FUNCTION_BLOCK Spreader EXTENDS OperationalParticleSet
  VAR
    lSpuriousLoweredEndAB : SpuriousLoweredEnd;
    lSpuriousLoweredEndCD : SpuriousLoweredEnd;
    lTwistlocksReadyState : BOOL;
    lTwistlocksReadyStateCandidate : BOOL;
    lTwistlocksCurrentState : t_lock_state;
    lTwistlocksCurrentStateCandidate : t_lock_state;
    lTwistlocksEnabled : BOOL;
    lTwistlocksEnabledCandidate : BOOL;
    lTwistlockACurrentState : t_lock_state;
    lTwistlockALoweredState : ValueObjectBool;
    lTwistlockAReadyState : BOOL;
    lTwistlockACurrentStateCandidate : t_lock_state;
    lTwistlockALoweredStateCandidate : BOOL;
    lTwistlockAReadyStateCandidate : BOOL;
    lTwistlockBCurrentState : t_lock_state;
    lTwistlockBLoweredState : ValueObjectBool;
    lTwistlockBReadyState : BOOL;
    lTwistlockBCurrentStateCandidate : t_lock_state;
    lTwistlockBLoweredStateCandidate : BOOL;
    lTwistlockBReadyStateCandidate : BOOL;
    lTwistlockCCurrentState : t_lock_state;
    lTwistlockCLoweredState : ValueObjectBool;
    lTwistlockCReadyState : BOOL;
    lTwistlockCCurrentStateCandidate : t_lock_state;
    lTwistlockCLoweredStateCandidate : BOOL;
    lTwistlockCReadyStateCandidate : BOOL;
    lTwistlockDCurrentState : t_lock_state;
    lTwistlockDLoweredState : ValueObjectBool;
    lTwistlockDReadyState : BOOL;
    lTwistlockDCurrentStateCandidate : t_lock_state;
    lTwistlockDLoweredStateCandidate : BOOL;
    lTwistlockDReadyStateCandidate : BOOL;
  END_VAR

            ;
          

METHOD initialize
                  lSpuriousLoweredEndAB.Name := 'AB';
lSpuriousLoweredEndAB.Context REF= gSystemApollo.Lift.InputObject;
lSpuriousLoweredEndAB.PositionA REF= gSystemApollo.CANOpenMasterDriveApollo.WinchAngleA.PositionObject;
lSpuriousLoweredEndAB.PositionB REF= gSystemApollo.CANOpenMasterDriveApollo.WinchAngleB.PositionObject;
lSpuriousLoweredEndAB.TwistlockALoweredState REF= lTwistlockALoweredState;
lSpuriousLoweredEndAB.TwistlockALoweredStateCandidate REF= lTwistlockALoweredStateCandidate;
lSpuriousLoweredEndAB.TwistlockBLoweredState REF= lTwistlockBLoweredState;
lSpuriousLoweredEndAB.TwistlockBLoweredStateCandidate REF= lTwistlockBLoweredStateCandidate;
registerOperational(ADR(lSpuriousLoweredEndAB));

lSpuriousLoweredEndCD.Name := 'CD';
lSpuriousLoweredEndCD.Context REF= gSystemApollo.Lift.InputObject;
lSpuriousLoweredEndCD.PositionA REF= gSystemApollo.CANOpenMasterDriveApollo.WinchAngleC.PositionObject;
lSpuriousLoweredEndCD.PositionB REF= gSystemApollo.CANOpenMasterDriveApollo.WinchAngleD.PositionObject;
lSpuriousLoweredEndCD.TwistlockALoweredState REF= lTwistlockCLoweredState;
lSpuriousLoweredEndCD.TwistlockALoweredStateCandidate REF= lTwistlockCLoweredStateCandidate;
lSpuriousLoweredEndCD.TwistlockBLoweredState REF= lTwistlockDLoweredState;
lSpuriousLoweredEndCD.TwistlockBLoweredStateCandidate REF= lTwistlockDLoweredStateCandidate;
registerOperational(ADR(lSpuriousLoweredEndCD));

lTwistlockALoweredState.initializeValueObjectOp(OpSelf,'TwstALow','Twistlock A lowered','',cValueStyleConfigurable);
lTwistlockBLoweredState.initializeValueObjectOp(OpSelf,'TwstBLow','Twistlock B lowered','',cValueStyleConfigurable);
lTwistlockCLoweredState.initializeValueObjectOp(OpSelf,'TwstCLow','Twistlock C lowered','',cValueStyleConfigurable);
lTwistlockDLoweredState.initializeValueObjectOp(OpSelf,'TwstDLow','Twistlock D lowered','',cValueStyleConfigurable);

SUPER^.initialize();
SubSystem := cSubsystemSpreader;

                
END_METHOD

METHOD operator
                  lTwistlockACurrentStateCandidate := gSystemApollo.CANOpenMasterDriveApollo.Spreader.TwistlockACurrentState;
lTwistlockALoweredStateCandidate := gSystemApollo.CANOpenMasterDriveApollo.Spreader.TwistlockALoweredState;
lTwistlockAReadyStateCandidate := gSystemApollo.CANOpenMasterDriveApollo.Spreader.TwistlockAReadyState;

lTwistlockACurrentState := lTwistlockACurrentStateCandidate;
lTwistlockALoweredState.Value := lTwistlockALoweredStateCandidate;
lTwistlockAReadyState := lTwistlockAReadyStateCandidate;

lTwistlockBCurrentStateCandidate := gSystemApollo.CANOpenMasterDriveApollo.Spreader.TwistlockBCurrentState;
lTwistlockBLoweredStateCandidate := gSystemApollo.CANOpenMasterDriveApollo.Spreader.TwistlockBLoweredState;
lTwistlockBReadyStateCandidate := gSystemApollo.CANOpenMasterDriveApollo.Spreader.TwistlockBReadyState;

lTwistlockBCurrentState := lTwistlockBCurrentStateCandidate;
lTwistlockBLoweredState.Value := lTwistlockBLoweredStateCandidate;
lTwistlockBReadyState := lTwistlockBReadyStateCandidate;

lTwistlockCCurrentStateCandidate := gSystemApollo.CANOpenMasterDriveApollo.Spreader.TwistlockCCurrentState;
lTwistlockCLoweredStateCandidate := gSystemApollo.CANOpenMasterDriveApollo.Spreader.TwistlockCLoweredState;
lTwistlockCReadyStateCandidate := gSystemApollo.CANOpenMasterDriveApollo.Spreader.TwistlockCReadyState;

lTwistlockCCurrentState := lTwistlockCCurrentStateCandidate;
lTwistlockCLoweredState.Value := lTwistlockCLoweredStateCandidate;
lTwistlockCReadyState := lTwistlockCReadyStateCandidate;

lTwistlockDCurrentStateCandidate := gSystemApollo.CANOpenMasterDriveApollo.Spreader.TwistlockDCurrentState;
lTwistlockDLoweredStateCandidate := gSystemApollo.CANOpenMasterDriveApollo.Spreader.TwistlockDLoweredState;
lTwistlockDReadyStateCandidate := gSystemApollo.CANOpenMasterDriveApollo.Spreader.TwistlockDReadyState;

lTwistlockDCurrentState := lTwistlockDCurrentStateCandidate;
lTwistlockDLoweredState.Value := lTwistlockDLoweredStateCandidate;
lTwistlockDReadyState := lTwistlockDReadyStateCandidate;

lTwistlocksReadyStateCandidate := gSystemApollo.CANOpenMasterDriveApollo.Spreader.TwistlocksReadyState;
lTwistlocksReadyState := lTwistlocksReadyStateCandidate;

lTwistlocksCurrentStateCandidate := gSystemApollo.CANOpenMasterDriveApollo.Spreader.TwistlocksCurrentState;
lTwistlocksCurrentState := lTwistlocksCurrentStateCandidate;
IF (lTwistlocksCurrentState=t_lock_state.cLockStateNone) THEN
	lTwistlocksCurrentState := t_lock_state.cLockStatePartial;
END_IF

SUPER^.operator();

lTwistlocksEnabledCandidate := gSystemApollo.CANOpenMasterDriveApollo.Spreader.TwistlocksEnabled;
lTwistlocksEnabled := ((lTwistlocksEnabledCandidate) OR
	((lTwistlockALoweredState.Value) AND
	(lTwistlockBLoweredState.Value) AND
	(lTwistlockCLoweredState.Value) AND
	(lTwistlockDLoweredState.Value)));
		
                
END_METHOD

PROPERTY TwistlockACurrentState : t_lock_state
GET
                    TwistlockACurrentState := lTwistlockACurrentState;

                  
END_GET
END_PROPERTY

PROPERTY TwistlockALoweredState : BOOL
GET
                    TwistlockALoweredState := lTwistlockALoweredState.Value;

                  
END_GET
END_PROPERTY

PROPERTY TwistlockALoweredStateObject : REFERENCE TO ValueObjectBool
GET
                    TwistlockALoweredStateObject REF= lTwistlockALoweredState;

                  
END_GET
END_PROPERTY

PROPERTY TwistlockAReadyState : BOOL
GET
                    TwistlockAReadyState := lTwistlockAReadyState;

                  
END_GET
END_PROPERTY

PROPERTY TwistlockBCurrentState : t_lock_state
GET
                    TwistlockBCurrentState := lTwistlockBCurrentState;

                  
END_GET
END_PROPERTY

PROPERTY TwistlockBLoweredState : BOOL
GET
                    TwistlockBLoweredState := lTwistlockBLoweredState.Value;

                  
END_GET
END_PROPERTY

PROPERTY TwistlockBLoweredStateObject : REFERENCE TO ValueObjectBool
GET
                    TwistlockBLoweredStateObject REF= lTwistlockBLoweredState;

                  
END_GET
END_PROPERTY

PROPERTY TwistlockBReadyState : BOOL
GET
                    TwistlockBReadyState := lTwistlockBReadyState;

                  
END_GET
END_PROPERTY

PROPERTY TwistlockCCurrentState : t_lock_state
GET
                    TwistlockCCurrentState := lTwistlockCCurrentState;

                  
END_GET
END_PROPERTY

PROPERTY TwistlockCLoweredState : BOOL
GET
                    TwistlockCLoweredState := lTwistlockCLoweredState.Value;

                  
END_GET
END_PROPERTY

PROPERTY TwistlockCLoweredStateObject : REFERENCE TO ValueObjectBool
GET
                    TwistlockCLoweredStateObject REF= lTwistlockCLoweredState;

                  
END_GET
END_PROPERTY

PROPERTY TwistlockCReadyState : BOOL
GET
                    TwistlockCReadyState := lTwistlockCReadyState;

                  
END_GET
END_PROPERTY

PROPERTY TwistlockDCurrentState : t_lock_state
GET
                    TwistlockDCurrentState := lTwistlockDCurrentState;

                  
END_GET
END_PROPERTY

PROPERTY TwistlockDLoweredState : BOOL
GET
                    TwistlockDLoweredState := lTwistlockDLoweredState.Value;

                  
END_GET
END_PROPERTY

PROPERTY TwistlockDLoweredStateObject : REFERENCE TO ValueObjectBool
GET
                    TwistlockDLoweredStateObject REF= lTwistlockDLoweredState;

                  
END_GET
END_PROPERTY

PROPERTY TwistlockDReadyState : BOOL
GET
                    TwistlockDReadyState := lTwistlockDReadyState;

                  
END_GET
END_PROPERTY

PROPERTY TwistlocksCurrentState : t_lock_state
GET
                    TwistlocksCurrentState := lTwistlocksCurrentState;

                  
END_GET
END_PROPERTY

PROPERTY TwistlocksEnabled : BOOL
GET
                    TwistlocksEnabled := lTwistlocksEnabled;

                  
END_GET
END_PROPERTY

PROPERTY TwistlocksReadyState : BOOL
GET
                    TwistlocksReadyState := lTwistlocksReadyState;

                  
END_GET
END_PROPERTY

PROPERTY TypeToken : t_medium_string
GET
                    TypeToken := 'Spreader';
                  
END_GET
END_PROPERTY
END_FUNCTION_BLOCK

FUNCTION_BLOCK SpuriousLoweredEnd EXTENDS NonOperationalParticleSet
  VAR
    lEnable : BOOL := TRUE;
    lContext : REFERENCE TO ValueObjectPercentage;
    lPositionA : REFERENCE TO ValueObjectPercentage;
    lPositionB : REFERENCE TO ValueObjectPercentage;
    lPositionLimit : t_percentage := 0.05;  (* machine height dependent *)
    lContextReset : t_percentage := 0.05;
    lPosition : t_percentage;
    lResetPosition : t_percentage;
    lAllowAdditionalMovement : BOOL;
    lTwistlockALoweredState : REFERENCE TO ValueObjectBool;
    lTwistlockALoweredStateCandidate : REFERENCE TO BOOL;
    lTwistlockBLoweredState : REFERENCE TO ValueObjectBool;
    lTwistlockBLoweredStateCandidate : REFERENCE TO BOOL;
  END_VAR

            ;
          

METHOD operator
                  SUPER^.operator();

IF (NOT(lEnable)) THEN
	RETURN;
END_IF

// robustness measures:
// traveling and one false/on (sensor false positive or container moves): masked until lowered to limit, further upon context reset
// lowering and one false/off (sensor fails to detect): allows further lowering to limit, warning as further upon context reset possible
// lowered but chassis/stack movement or signaled too early or pulse raised: masked until lowered to limit

// average is considered more robust than per corner specific 
lPosition := (lPositionA.Value + lPositionB.Value) / 2.0;

// foobar error handling notification

IF ((lTwistlockALoweredStateCandidate) AND (lTwistlockBLoweredStateCandidate)) THEN
	lAllowAdditionalMovement := ((lResetPosition - lPosition) < lPositionLimit);

	lTwistlockALoweredState.Value := NOT(lAllowAdditionalMovement);
	lTwistlockBLoweredState.Value := NOT(lAllowAdditionalMovement);

	RETURN;
END_IF
	
IF (((NOT(lTwistlockALoweredStateCandidate)) AND (lTwistlockBLoweredStateCandidate)) OR	
	((NOT(lTwistlockBLoweredStateCandidate)) AND (lTwistlockALoweredStateCandidate))) THEN
	IF (lContext.Value>=lContextReset) THEN		
		lResetPosition := lPosition;
	END_IF

	lAllowAdditionalMovement := ((lResetPosition - lPosition) < lPositionLimit);

	lTwistlockALoweredState.Value := NOT(lAllowAdditionalMovement);
	lTwistlockBLoweredState.Value := NOT(lAllowAdditionalMovement);
	
	RETURN;
END_IF

lResetPosition := lPosition;

lTwistlockALoweredState.Value := lTwistlockALoweredStateCandidate;
lTwistlockBLoweredState.Value := lTwistlockBLoweredStateCandidate;

                
END_METHOD

PROPERTY Context : REFERENCE TO ValueObjectPercentage
GET
                    Context ref= lContext;
                  
END_GET
SET
                    lContext ref= Context;
                  
END_SET
END_PROPERTY

PROPERTY ContextReset : t_percentage
GET
                    ContextReset := lContextReset;
                  
END_GET
SET
                    lContextReset := ContextReset;
                  
END_SET
END_PROPERTY

PROPERTY PositionA : REFERENCE TO ValueObjectPercentage
GET
                    PositionA ref= lPositionA;
                  
END_GET
SET
                    lPositionA ref= PositionA;
                  
END_SET
END_PROPERTY

PROPERTY PositionB : REFERENCE TO ValueObjectPercentage
GET
                    PositionB ref= lPositionB;
                  
END_GET
SET
                    lPositionB ref= PositionB;
                  
END_SET
END_PROPERTY

PROPERTY PositionLimit : t_percentage
GET
                    PositionLimit := lPositionLimit;
                  
END_GET
SET
                    lPositionLimit := PositionLimit;
                  
END_SET
END_PROPERTY

PROPERTY TwistlockALoweredState : REFERENCE TO ValueObjectBool
SET
                    lTwistlockALoweredState ref= TwistlockALoweredState;
                  
END_SET
END_PROPERTY

PROPERTY TwistlockALoweredStateCandidate : REFERENCE TO BOOL
SET
                    lTwistlockALoweredStateCandidate ref= TwistlockALoweredStateCandidate;
                  
END_SET
END_PROPERTY

PROPERTY TwistlockBLoweredState : REFERENCE TO ValueObjectBool
SET
                    lTwistlockBLoweredState ref= TwistlockBLoweredState;
                  
END_SET
END_PROPERTY

PROPERTY TwistlockBLoweredStateCandidate : REFERENCE TO BOOL
SET
                    lTwistlockBLoweredStateCandidate ref= TwistlockBLoweredStateCandidate;
                  
END_SET
END_PROPERTY

PROPERTY TypeToken : t_medium_string
GET
                    TypeToken := 'SpreaderFilter';
                  
END_GET
END_PROPERTY
END_FUNCTION_BLOCK

FUNCTION_BLOCK UIEventApollo EXTENDS UIEvent

            ;
          

METHOD _operator
                  SUPER^._operator();

CASE lUIEventCode OF
	cUIEventCodeToggleSpreaderConfiguration:
		gSystemApollo.CANOpenMasterDriveApollo.Spreader.TelescopingEnableCommand := TRUE;

	cUIEventCodeSpreaderExtensionAutoCommand:
		gSystemApollo.CANOpenMasterDriveApollo.Spreader.TelescopingExtendAutoCommand := TRUE;
	
	cUIEventCodeSpreaderRetractionAutoCommand:
		gSystemApollo.CANOpenMasterDriveApollo.Spreader.TelescopingRetractAutoCommand := TRUE;
END_CASE

                
END_METHOD
END_FUNCTION_BLOCK

FUNCTION_BLOCK UInterfaceCabinApollo EXTENDS UInterfaceCabin
  VAR
    lPackSystem : PackSystemPLC;
    lPackMovement : PackMovementPLCApollo;
    lPackReportable : PackReportablePLC;
    lPackSpreader : PackSpreaderPLC;
    lPackUICommand : PackUICommandPLC;
  END_VAR

            ;
          

METHOD initializeUInterfaceCabinApollo
  VAR_INPUT
    packProvider : REFERENCE TO PackProvider;
    reportableChannelUIR : REFERENCE TO ReportableChannelUIR;
  END_VAR
                  lPackSystem.initializePackSystemPLC(THIS^);
lPackUICommand.initializePackUICommandPLC(THIS^);
lPackReportable.initializePackReportablePLC(reportableChannelUIR);

initializeUInterfacePLC(lPackSystem,
	lPackMovement,
	lPackReportable,
	lPackSpreader,
	lPackUICommand,
	packProvider);

                
END_METHOD
END_FUNCTION_BLOCK

FUNCTION_BLOCK UInterfaceDualRadioCabin EXTENDS UInterfaceDual
  VAR
    lUInterfaceRadio : UInterfaceRadioApollo;
    lUInterfaceCabin : UInterfaceCabinApollo;
  END_VAR

            ;
          

METHOD initialize
                  UInterfaceA REF= lUInterfaceRadio;
UInterfaceB REF= lUInterfaceCabin;

registerNonOperational(ADR(lUInterfaceRadio));
registerNonOperational(ADR(lUInterfaceCabin));

SUPER^.initialize();

lUInterfaceRadio.UInterfaceId := t_ui_id.cUIIdA;
lUInterfaceCabin.UInterfaceId := t_ui_id.cUIIdB;


                
END_METHOD

PROPERTY SlowFactor : REAL
SET
                    UInterfaceRadio.SlowFactor := SlowFactor;
//UInterfaceCabin.SlowFactor := SlowFactor;
                  
END_SET
END_PROPERTY

PROPERTY TypeToken : t_medium_string
GET
                    TypeToken := 'UIRadioCabin';
                  
END_GET
END_PROPERTY

PROPERTY UInterfaceCabin : REFERENCE TO UInterfaceCabinApollo
GET
                    UInterfaceCabin ref= lUInterfaceCabin;
                  
END_GET
END_PROPERTY

PROPERTY UInterfaceRadio : REFERENCE TO UInterfaceRadioApollo
GET
                    UInterfaceRadio ref= lUInterfaceRadio;
                  
END_GET
END_PROPERTY
END_FUNCTION_BLOCK

FUNCTION_BLOCK PackMovementPLCApollo EXTENDS PackMovementPLC

            
          

METHOD read
                  SUPER^.read();

lLiftABPosition := (gSystemApollo.CANOpenMasterDriveApollo.WinchAngleA.Position + gSystemApollo.CANOpenMasterDriveApollo.WinchAngleB.Position)/2.0;
lLiftCDPosition := (gSystemApollo.CANOpenMasterDriveApollo.WinchAngleC.Position + gSystemApollo.CANOpenMasterDriveApollo.WinchAngleD.Position)/2.0;

                
END_METHOD
END_FUNCTION_BLOCK

FUNCTION_BLOCK PackSpreaderPLC EXTENDS PackSpreader

            
          

METHOD read
                  lSideShiftActive := ((gSystemApollo.SystemState.State=cSystemStateOperational) AND
	((gSystemApollo.CANOpenMasterDriveApollo.Spreader.SideshiftABCommand<>0.0) OR
	(gSystemApollo.CANOpenMasterDriveApollo.Spreader.SideshiftCDCommand<>0.0)));

lTwistlocksState := gSystemApollo.Spreader.TwistlocksCurrentState;

lStateA := gSystemApollo.CANOpenMasterDriveApollo.Spreader.TwistlockACurrentState;
lLoweredA := gSystemApollo.CANOpenMasterDriveApollo.Spreader.TwistlockALoweredState;
lStateB := gSystemApollo.CANOpenMasterDriveApollo.Spreader.TwistlockBCurrentState;
lLoweredB := gSystemApollo.CANOpenMasterDriveApollo.Spreader.TwistlockBLoweredState;
lStateC := gSystemApollo.CANOpenMasterDriveApollo.Spreader.TwistlockCCurrentState;
lLoweredC := gSystemApollo.CANOpenMasterDriveApollo.Spreader.TwistlockCLoweredState;
lStateD := gSystemApollo.CANOpenMasterDriveApollo.Spreader.TwistlockDCurrentState;
lLoweredD := gSystemApollo.CANOpenMasterDriveApollo.Spreader.TwistlockDLoweredState;

lExtensionState := t_spreader_extension_state.cSpreaderExtensionState6m;

lSpreaderOperationEnabled := gSystemApollo.Spreader.TwistlocksEnabled;
lSpreaderOperationActive := ((gSystemApollo.Spreader.TwistlockALoweredState) OR
	(gSystemApollo.Spreader.TwistlockBLoweredState) OR
	(gSystemApollo.Spreader.TwistlockCLoweredState) OR
	(gSystemApollo.Spreader.TwistlockDLoweredState));

lSpreaderConfigurationOptionEnabled := ((gSystemPrimary.SystemState.State=cSystemStateOperational) AND
	(gSystemApollo.OperatingMode.Mode>cOperatingModeUnparking) AND
	(lTwistlocksState=cLockStateUnlocked) AND
	(NOT(lLoweredA)) AND
	(NOT(lLoweredB)) AND
	(NOT(lLoweredC)) AND
	(NOT(lLoweredD)));
lSpreaderConfigurationEnabled := gSystemApollo.CANOpenMasterDriveApollo.Spreader.TelescopingEnabled;
lSpreaderConfigurationActive := gSystemApollo.CANOpenMasterDriveApollo.Spreader.TelescopingActive;
lSpreaderConfigurationExtending := ((gSystemApollo.CANOpenMasterDriveApollo.Spreader.TelescopingActive) AND (gSystemApollo.CANOpenMasterDriveApollo.Spreader.TelescopingExtendCommand));
lSpreaderConfigurationRetracting := ((gSystemApollo.CANOpenMasterDriveApollo.Spreader.TelescopingActive) AND (gSystemApollo.CANOpenMasterDriveApollo.Spreader.TelescopingRetractCommand));

	
                
END_METHOD
END_FUNCTION_BLOCK

FUNCTION_BLOCK UInterfaceDualRadio EXTENDS UInterfaceDual
  VAR
    lUInterfaceRadioA : UInterfaceRadioApollo;
    lUInterfaceRadioB : UInterfaceRadioApollo;
  END_VAR

            ;
          

METHOD initialize
                  UInterfaceA REF= lUInterfaceRadioA;
UInterfaceB REF= lUInterfaceRadioB;

lUInterfaceRadioA.Name := 'RadioA';
registerNonOperational(ADR(lUInterfaceRadioA));

lUInterfaceRadioB.Name := 'RadioB';
registerNonOperational(ADR(lUInterfaceRadioB));

SUPER^.initialize();

lUInterfaceRadioA.UInterfaceId := t_ui_id.cUIIdA;
lUInterfaceRadioB.UInterfaceId := t_ui_id.cUIIdB;
                
END_METHOD

PROPERTY SlowFactor : REAL
SET
                    UInterfaceRadioA.SlowFactor := SlowFactor;
UInterfaceRadioB.SlowFactor := SlowFactor;
                  
END_SET
END_PROPERTY

PROPERTY TypeToken : t_medium_string
GET
                    TypeToken := 'UIRadioRadio';
                  
END_GET
END_PROPERTY

PROPERTY UInterfaceRadioA : REFERENCE TO UInterfaceRadioApollo
GET
                    UInterfaceRadioA ref= lUInterfaceRadioA;
                  
END_GET
END_PROPERTY

PROPERTY UInterfaceRadioB : REFERENCE TO UInterfaceRadioApollo
GET
                    UInterfaceRadioB ref= lUInterfaceRadioB;
                  
END_GET
END_PROPERTY
END_FUNCTION_BLOCK

FUNCTION_BLOCK UInterfaceRadioApollo EXTENDS UInterfaceRadio
  VAR
    lPackSystem : PackSystemPLC;
    lPackMovement : PackMovementPLCApollo;
    lPackReportable : PackReportablePLC;
    lPackSpreader : PackSpreaderPLC;
    lPackUICommand : PackUICommandPLC;
  END_VAR

            ;
          

METHOD initializelUInterfaceRadioApollo
  VAR_INPUT
    packProvider : REFERENCE TO PackProvider;
    reportableChannelUIR : REFERENCE TO ReportableChannelUIR;
  END_VAR
                  lPackSystem.initializePackSystemPLC(THIS^);
lPackUICommand.initializePackUICommandPLC(THIS^);
lPackReportable.initializePackReportablePLC(reportableChannelUIR);

initializeUInterfacePLC(lPackSystem,
	lPackMovement,
	lPackReportable,
	lPackSpreader,
	lPackUICommand,
	packProvider);


                
END_METHOD
END_FUNCTION_BLOCK
